PROGRAM MAIN
VAR
    gatewaySmokeTests : FB_GatewaySmokeTests;
END_VAR

TcUnit.RUN();

END_PROGRAM

(* stored: Version 1.1.0.1, ProductVersion 3.1.4024.9
   POU MAIN: Id {b72daeb9-f97b-498a-8662-597d8e37f5bc}, SpecialFunc None *)
